  MoveAbsJ [[1.70,5.99,18.89,159.17,24.55,90.17],[9E9,9E9,9E9,9E9,9E9,9E9]],speeddata0,DefaultBlend,tool0;
  MoveAbsJ [[1.62,6.16,19.16,160.16,25.01,90.16],[9E9,9E9,9E9,9E9,9E9,9E9]],speeddata0,DefaultBlend,tool0;
  MoveAbsJ [[1.54,6.32,19.44,161.15,25.47,90.15],[9E9,9E9,9E9,9E9,9E9,9E9]],speeddata0,DefaultBlend,tool0;
  MoveAbsJ [[1.45,6.49,19.71,162.14,25.93,90.15],[9E9,9E9,9E9,9E9,9E9,9E9]],speeddata0,DefaultBlend,tool0;
  MoveAbsJ [[1.37,6.66,19.99,163.14,26.38,90.14],[9E9,9E9,9E9,9E9,9E9,9E9]],speeddata0,DefaultBlend,tool0;
  MoveAbsJ [[1.29,6.83,20.26,164.13,26.84,90.13],[9E9,9E9,9E9,9E9,9E9,9E9]],speeddata0,DefaultBlend,tool0;
  MoveAbsJ [[1.21,6.99,20.54,165.12,27.30,90.13],[9E9,9E9,9E9,9E9,9E9,9E9]],speeddata0,DefaultBlend,tool0;
  MoveAbsJ [[1.13,7.16,20.81,166.11,27.76,90.12],[9E9,9E9,9E9,9E9,9E9,9E9]],speeddata0,DefaultBlend,tool0;
  MoveAbsJ [[1.05,7.33,21.08,167.10,28.21,90.11],[9E9,9E9,9E9,9E9,9E9,9E9]],speeddata0,DefaultBlend,tool0;
  MoveAbsJ [[0.97,7.50,21.36,168.09,28.67,90.10],[9E9,9E9,9E9,9E9,9E9,9E9]],speeddata0,DefaultBlend,tool0;
  MoveAbsJ [[0.89,7.66,21.63,169.08,29.13,90.10],[9E9,9E9,9E9,9E9,9E9,9E9]],speeddata0,DefaultBlend,tool0;
  MoveAbsJ [[0.80,7.83,21.91,170.07,29.59,90.09],[9E9,9E9,9E9,9E9,9E9,9E9]],speeddata0,DefaultBlend,tool0;
  MoveAbsJ [[0.72,8.00,22.18,171.06,30.04,90.08],[9E9,9E9,9E9,9E9,9E9,9E9]],speeddata0,DefaultBlend,tool0;
  MoveAbsJ [[0.64,8.17,22.46,172.05,30.50,90.07],[9E9,9E9,9E9,9E9,9E9,9E9]],speeddata0,DefaultBlend,tool0;
  MoveAbsJ [[0.56,8.33,22.73,173.04,30.96,90.07],[9E9,9E9,9E9,9E9,9E9,9E9]],speeddata0,DefaultBlend,tool0;
  MoveAbsJ [[0.48,8.50,23.01,174.04,31.42,90.06],[9E9,9E9,9E9,9E9,9E9,9E9]],speeddata0,DefaultBlend,tool0;
  MoveAbsJ [[0.40,8.67,23.28,175.03,31.87,90.05],[9E9,9E9,9E9,9E9,9E9,9E9]],speeddata0,DefaultBlend,tool0;
  MoveAbsJ [[0.32,8.84,23.56,176.02,32.33,90.05],[9E9,9E9,9E9,9E9,9E9,9E9]],speeddata0,DefaultBlend,tool0;
  MoveAbsJ [[0.24,9.00,23.83,177.01,32.79,90.04],[9E9,9E9,9E9,9E9,9E9,9E9]],speeddata0,DefaultBlend,tool0;
  MoveAbsJ [[0.15,9.17,24.11,178.00,33.25,90.03],[9E9,9E9,9E9,9E9,9E9,9E9]],speeddata0,DefaultBlend,tool0;
  MoveAbsJ [[0.07,9.34,24.38,178.99,33.71,90.02],[9E9,9E9,9E9,9E9,9E9,9E9]],speeddata0,DefaultBlend,tool0;
  MoveAbsJ [[-0.01,9.51,24.66,179.98,34.16,90.02],[9E9,9E9,9E9,9E9,9E9,9E9]],speeddata0,FinePoint,tool0;
  TPWrite "Action 53 LinearMovement.";
  MoveAbsJ [[-0.01,9.51,24.66,179.98,34.16,90.02],[9E9,9E9,9E9,9E9,9E9,9E9]],speeddata0,DefaultBlend,tool0;
  MoveAbsJ [[-0.00,9.97,25.29,180.00,35.26,90.00],[9E9,9E9,9E9,9E9,9E9,9E9]],speeddata0,DefaultBlend,tool0;
  MoveAbsJ [[-0.00,10.45,25.94,180.00,36.38,90.00],[9E9,9E9,9E9,9E9,9E9,9E9]],speeddata0,DefaultBlend,tool0;
  MoveAbsJ [[-0.00,10.95,26.56,180.00,37.51,90.00],[9E9,9E9,9E9,9E9,9E9,9E9]],speeddata0,DefaultBlend,tool0;
  MoveAbsJ [[-0.00,11.47,27.16,180.00,38.63,90.00],[9E9,9E9,9E9,9E9,9E9,9E9]],speeddata0,DefaultBlend,tool0;
  MoveAbsJ [[-0.00,12.02,27.74,180.00,39.76,90.00],[9E9,9E9,9E9,9E9,9E9,9E9]],speeddata0,DefaultBlend,tool0;
  MoveAbsJ [[-0.00,12.59,28.29,180.00,40.88,90.00],[9E9,9E9,9E9,9E9,9E9,9E9]],speeddata0,DefaultBlend,tool0;
  MoveAbsJ [[-0.00,13.18,28.83,180.00,42.01,90.00],[9E9,9E9,9E9,9E9,9E9,9E9]],speeddata0,DefaultBlend,tool0;
  MoveAbsJ [[-0.00,13.80,29.33,180.00,43.13,90.00],[9E9,9E9,9E9,9E9,9E9,9E9]],speeddata0,FinePoint,tool0;
  TPWrite "Action 54 OpenGripper.";
  TPWrite "Press Play to Continue";
  Stop;
  TPWrite "Action 55 LinearMovement.";
  MoveAbsJ [[-0.00,13.80,29.34,180.00,43.14,90.00],[9E9,9E9,9E9,9E9,9E9,9E9]],speeddata0,DefaultBlend,tool0;
  MoveAbsJ [[-0.00,12.74,30.66,180.00,43.39,90.00],[9E9,9E9,9E9,9E9,9E9,9E9]],speeddata0,DefaultBlend,tool0;
  MoveAbsJ [[-0.00,11.64,32.01,180.00,43.64,90.00],[9E9,9E9,9E9,9E9,9E9,9E9]],speeddata0,DefaultBlend,tool0;
  MoveAbsJ [[-0.00,10.53,33.34,180.00,43.87,90.00],[9E9,9E9,9E9,9E9,9E9,9E9]],speeddata0,DefaultBlend,tool0;
  MoveAbsJ [[-0.00,9.42,34.66,180.00,44.08,90.00],[9E9,9E9,9E9,9E9,9E9,9E9]],speeddata0,DefaultBlend,tool0;
  MoveAbsJ [[-0.00,8.30,35.97,180.00,44.26,90.00],[9E9,9E9,9E9,9E9,9E9,9E9]],speeddata0,DefaultBlend,tool0;
  MoveAbsJ [[-0.00,7.17,37.26,180.00,44.43,90.00],[9E9,9E9,9E9,9E9,9E9,9E9]],speeddata0,DefaultBlend,tool0;
  MoveAbsJ [[-0.00,6.03,38.54,180.00,44.57,90.00],[9E9,9E9,9E9,9E9,9E9,9E9]],speeddata0,DefaultBlend,tool0;
  MoveAbsJ [[0.00,4.88,39.81,180.00,44.69,90.00],[9E9,9E9,9E9,9E9,9E9,9E9]],speeddata0,FinePoint,tool0;
  !Move back to Initial Config at the end
  MoveAbsJ TGofa_InitialConfig,speeddata0,FinePoint,tool0;
  TPWrite "Program Execution Complete";
EndProc

EndModule
